PROGRAM maint_mode
VAR
	maint_mode: BOOL;
	
	u_3112_hmi_start_request: BOOL;
	u_3112_maint_request: BOOL;
	u_3112_hmi_speed_request: REAL;
	u_3112_maint_speed_request: REAL;
	u_3112_hmi_stop_request: BOOL;
	
	u_3212_hmi_start_request: BOOL;
	u_3212_maint_request: BOOL;
	u_3212_hmi_speed_request: REAL;
	u_3212_maint_speed_request: REAL;
	u_3212_hmi_stop_request: BOOL;

	u_3312_hmi_start_request: BOOL;
	u_3312_maint_request: BOOL;
	u_3312_hmi_speed_request: REAL;
	u_3312_maint_speed_request: REAL;
	u_3312_hmi_stop_request: BOOL;
	
	u_3405_hmi_start_request: BOOL;
	u_3405_maint_request: BOOL;
	u_3405_hmi_speed_request: REAL;
	u_3405_maint_speed_request: REAL;
	u_3405_hmi_stop_request: BOOL;
	
	u_3160_hmi_start_request: BOOL;
	u_3160_maint_request: BOOL;
	u_3160_hmi_speed_request: REAL;
	u_3160_maint_speed_request: REAL;
	u_3160_hmi_stop_request: BOOL;
	
	u_3260_hmi_start_request: BOOL;
	u_3260_maint_request: BOOL;
	u_3260_hmi_speed_request: REAL;
	u_3260_maint_speed_request: REAL;
	u_3260_hmi_stop_request: BOOL;
	
	u_3360_hmi_start_request: BOOL;
	u_3360_maint_request: BOOL;
	u_3360_hmi_speed_request: REAL;
	u_3360_maint_speed_request: REAL;
	u_3360_hmi_stop_request: BOOL;
	
	nv_3110_hmi_open_request: BOOL;
	nv_3110_hmi_close_request: BOOL;
	nv_3110_maint_request: BOOL;
	
	nv_3210_hmi_open_request: BOOL;
	nv_3210_hmi_close_request: BOOL;
	nv_3210_maint_request: BOOL;
	
	nv_3310_hmi_open_request: BOOL;
	nv_3310_hmi_close_request: BOOL;
	nv_3310_maint_request: BOOL;
	
	nv_3135_hmi_open_request: BOOL;
	nv_3135_hmi_close_request: BOOL;
	nv_3135_maint_request: BOOL;
	
	nv_3235_hmi_open_request: BOOL;
	nv_3235_hmi_close_request: BOOL;
	nv_3235_maint_request: BOOL;
	
	nv_3335_hmi_open_request: BOOL;
	nv_3335_hmi_close_request: BOOL;
	nv_3335_maint_request: BOOL;
	
	nv_3372_hmi_open_request: BOOL;
	nv_3372_hmi_close_request: BOOL;
	nv_3372_maint_request: BOOL;
	u_3370_hmi_start_request: BOOL;
	u_3370_maint_request: BOOL;
	u_3370_hmi_stop_request: BOOL;
	u_3370_hmi_speed_request: REAL;
	u_3370_maint_speed_request: REAL;
	nv_3162_hmi_open_request: BOOL;
	nv_3162_maint_request: BOOL;
	nv_3162_hmi_close_request: BOOL;
END_VAR

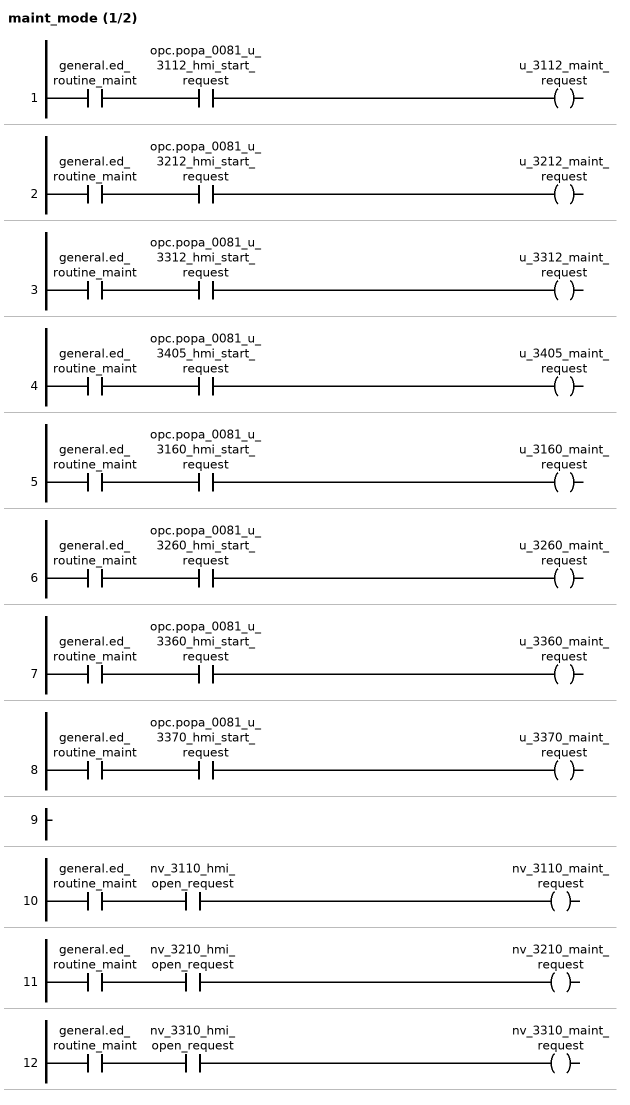
// NETWORK 1
u_3112_maint_request := general.ed_routine_maint AND opc.popa_0081_u_3112_hmi_start_request;

// NETWORK 2
u_3212_maint_request := general.ed_routine_maint AND opc.popa_0081_u_3212_hmi_start_request;

// NETWORK 3
u_3312_maint_request := general.ed_routine_maint AND opc.popa_0081_u_3312_hmi_start_request;

// NETWORK 4
u_3405_maint_request := general.ed_routine_maint AND opc.popa_0081_u_3405_hmi_start_request;

// NETWORK 5
u_3160_maint_request := general.ed_routine_maint AND opc.popa_0081_u_3160_hmi_start_request;

// NETWORK 6
u_3260_maint_request := general.ed_routine_maint AND opc.popa_0081_u_3260_hmi_start_request;

// NETWORK 7
u_3360_maint_request := general.ed_routine_maint AND opc.popa_0081_u_3360_hmi_start_request;

// NETWORK 8
u_3370_maint_request := general.ed_routine_maint AND opc.popa_0081_u_3370_hmi_start_request;

// NETWORK 9

// NETWORK 10
nv_3110_maint_request := general.ed_routine_maint AND nv_3110_hmi_open_request;

// NETWORK 11
nv_3210_maint_request := general.ed_routine_maint AND nv_3210_hmi_open_request;

// NETWORK 12
nv_3310_maint_request := general.ed_routine_maint AND nv_3310_hmi_open_request;

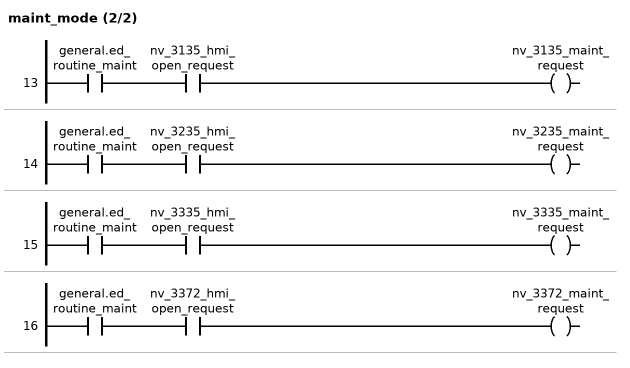
// NETWORK 13
nv_3135_maint_request := general.ed_routine_maint AND nv_3135_hmi_open_request;

// NETWORK 14
nv_3235_maint_request := general.ed_routine_maint AND nv_3235_hmi_open_request;

// NETWORK 15
nv_3335_maint_request := general.ed_routine_maint AND nv_3335_hmi_open_request;

// NETWORK 16
nv_3372_maint_request := general.ed_routine_maint AND nv_3372_hmi_open_request;

END_PROGRAM

(* stored: Version 1.1.0.1, ProductVersion 3.1.4024.12
   POU maint_mode: Id {fe91578f-e7b9-4e8e-a60b-a630302703f0}, SpecialFunc None *)
